// TIA Portal V21 export
TYPE "LBC_typeAnalogProcessValues"
TITLE = LBC_typeAnalogProcessValues
// Module related monitoring information
   STRUCT
      enable { ExternalWritable := 'False'} : Bool;   // Enable functionality of FB
      referenceDesignator { ExternalWritable := 'False'} : WString[154];   // Reference Designator for the module incl. its parent
      simulation { ExternalWritable := 'False'} : Bool;   // Enable simulation input of analog value
      processValue { ExternalWritable := 'False'} : LReal;   // Scaled process value
      analogValue { ExternalWritable := 'False'} : Int;   // Analog value for/from hardware periphery
      limitHigh2 { ExternalWritable := 'False'} : Bool;   // Process value limit high 2 exceeded (Lim 2 > Lim1, resets Lim 1)
      limitHigh1 { ExternalWritable := 'False'} : Bool;   // Process value limit high 1 exceeded
      limitLow1 { ExternalWritable := 'False'} : Bool;   // Process value limit low 1 exceeded
      limitLow2 { ExternalWritable := 'False'} : Bool;   // Process value limit low 2 exceeded (Lim 2 < Lim1, resets Lim 1)
      maxValueReached { ExternalWritable := 'False'} : Bool;   // Maximum configured process value reached. Value is limited to the maximum configured value.
      minValueReached { ExternalWritable := 'False'} : Bool;   // Minimum configured process value reached. Value is limited to the minimum configured value.
      error { ExternalWritable := 'False'} : Bool;   // An error occurred while processing the FB
      status { ExternalWritable := 'False'} : Word;   // 16#0000-16#7FFF: Status of the FB 16#8000-16#FFFF: Error identification
   END_STRUCT;
END_TYPE
